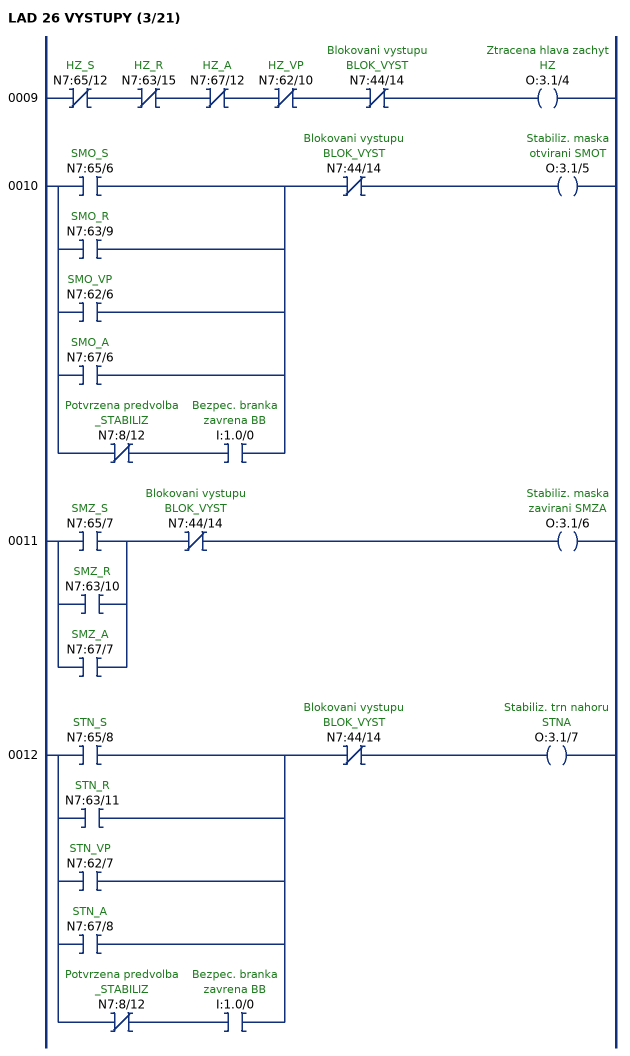
% Rung: 9 %
SOR XIO N7:65/12 XIO N7:63/15 XIO N7:67/12 XIO N7:62/10 XIO N7:44/14 OTE O:3.1/4 EOR
%   N7:65/12  HZ_S %
%   N7:63/15  HZ_R %
%   N7:67/12  HZ_A %
%   N7:62/10  HZ_VP %
%   N7:44/14  BLOK_VYST  "Blokovani vystupu" %
%   O:3.1/4  HZ  "Ztracena hlava zachyt" %
% Rung: 10 %
SOR BST XIC N7:65/6 NXB XIC N7:63/9 NXB XIC N7:62/6 NXB XIC N7:67/6 NXB XIO N7:8/12 XIC I:1.0/0 BND XIO N7:44/14 OTE O:3.1/5 EOR
%   N7:65/6  SMO_S %
%   N7:63/9  SMO_R %
%   N7:62/6  SMO_VP %
%   N7:67/6  SMO_A %
%   N7:8/12  _STABILIZ  "Potvrzena predvolba" %
%   I:1.0/0  BB  "Bezpec. branka zavrena" %
%   N7:44/14  BLOK_VYST  "Blokovani vystupu" %
%   O:3.1/5  SMOT  "Stabiliz. maska otvirani" %
% Rung: 11 %
SOR BST XIC N7:65/7 NXB XIC N7:63/10 NXB XIC N7:67/7 BND XIO N7:44/14 OTE O:3.1/6 EOR
%   N7:65/7  SMZ_S %
%   N7:63/10  SMZ_R %
%   N7:67/7  SMZ_A %
%   N7:44/14  BLOK_VYST  "Blokovani vystupu" %
%   O:3.1/6  SMZA  "Stabiliz. maska zavirani" %
% Rung: 12 %
SOR BST XIC N7:65/8 NXB XIC N7:63/11 NXB XIC N7:62/7 NXB XIC N7:67/8 NXB XIO N7:8/12 XIC I:1.0/0 BND XIO N7:44/14 OTE O:3.1/7 EOR
%   N7:65/8  STN_S %
%   N7:63/11  STN_R %
%   N7:62/7  STN_VP %
%   N7:67/8  STN_A %
%   N7:8/12  _STABILIZ  "Potvrzena predvolba" %
%   I:1.0/0  BB  "Bezpec. branka zavrena" %
%   N7:44/14  BLOK_VYST  "Blokovani vystupu" %
%   O:3.1/7  STNA  "Stabiliz. trn nahoru" %

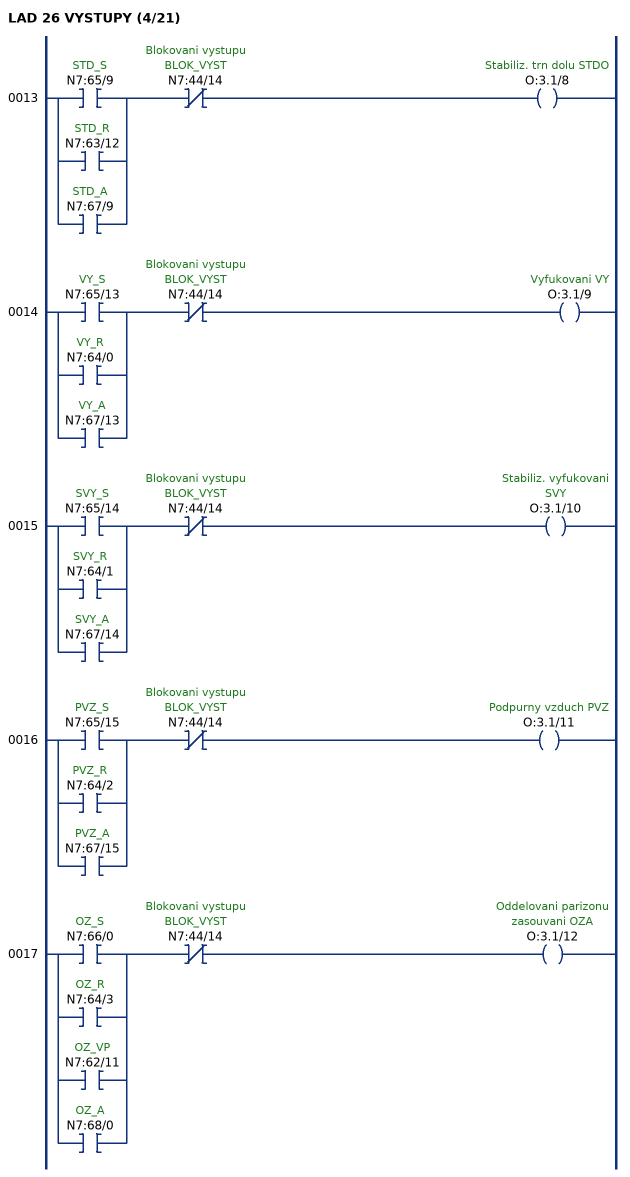
% Rung: 13 %
SOR BST XIC N7:65/9 NXB XIC N7:63/12 NXB XIC N7:67/9 BND XIO N7:44/14 OTE O:3.1/8 EOR
%   N7:65/9  STD_S %
%   N7:63/12  STD_R %
%   N7:67/9  STD_A %
%   N7:44/14  BLOK_VYST  "Blokovani vystupu" %
%   O:3.1/8  STDO  "Stabiliz. trn dolu" %
% Rung: 14 %
SOR BST XIC N7:65/13 NXB XIC N7:64/0 NXB XIC N7:67/13 BND XIO N7:44/14 OTE O:3.1/9 EOR
%   N7:65/13  VY_S %
%   N7:64/0  VY_R %
%   N7:67/13  VY_A %
%   N7:44/14  BLOK_VYST  "Blokovani vystupu" %
%   O:3.1/9  VY  "Vyfukovani" %
% Rung: 15 %
SOR BST XIC N7:65/14 NXB XIC N7:64/1 NXB XIC N7:67/14 BND XIO N7:44/14 OTE O:3.1/10 EOR
%   N7:65/14  SVY_S %
%   N7:64/1  SVY_R %
%   N7:67/14  SVY_A %
%   N7:44/14  BLOK_VYST  "Blokovani vystupu" %
%   O:3.1/10  SVY  "Stabiliz. vyfukovani" %
% Rung: 16 %
SOR BST XIC N7:65/15 NXB XIC N7:64/2 NXB XIC N7:67/15 BND XIO N7:44/14 OTE O:3.1/11 EOR
%   N7:65/15  PVZ_S %
%   N7:64/2  PVZ_R %
%   N7:67/15  PVZ_A %
%   N7:44/14  BLOK_VYST  "Blokovani vystupu" %
%   O:3.1/11  PVZ  "Podpurny vzduch" %
% Rung: 17 %
SOR BST XIC N7:66/0 NXB XIC N7:64/3 NXB XIC N7:62/11 NXB XIC N7:68/0 BND XIO N7:44/14 OTE O:3.1/12 EOR
%   N7:66/0  OZ_S %
%   N7:64/3  OZ_R %
%   N7:62/11  OZ_VP %
%   N7:68/0  OZ_A %
%   N7:44/14  BLOK_VYST  "Blokovani vystupu" %
%   O:3.1/12  OZA  "Oddelovani parizonu zasouvani" %

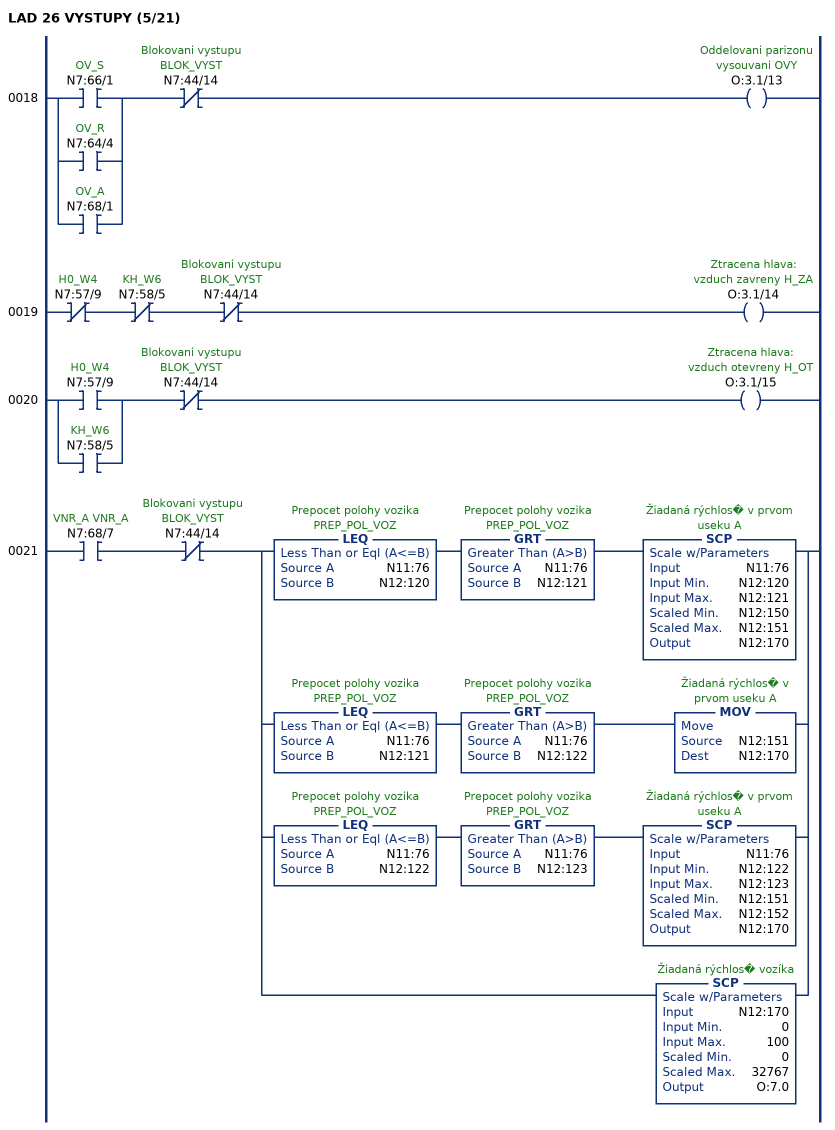
% Rung: 18 %
SOR BST XIC N7:66/1 NXB XIC N7:64/4 NXB XIC N7:68/1 BND XIO N7:44/14 OTE O:3.1/13 EOR
%   N7:66/1  OV_S %
%   N7:64/4  OV_R %
%   N7:68/1  OV_A %
%   N7:44/14  BLOK_VYST  "Blokovani vystupu" %
%   O:3.1/13  OVY  "Oddelovani parizonu vysouvani" %
% Rung: 19 %
SOR XIO N7:57/9 XIO N7:58/5 XIO N7:44/14 OTE O:3.1/14 EOR
%   N7:57/9  H0_W4 %
%   N7:58/5  KH_W6 %
%   N7:44/14  BLOK_VYST  "Blokovani vystupu" %
%   O:3.1/14  H_ZA  "Ztracena hlava: vzduch zavreny" %
% Rung: 20 %
SOR BST XIC N7:57/9 NXB XIC N7:58/5 BND XIO N7:44/14 OTE O:3.1/15 EOR
%   N7:57/9  H0_W4 %
%   N7:58/5  KH_W6 %
%   N7:44/14  BLOK_VYST  "Blokovani vystupu" %
%   O:3.1/15  H_OT  "Ztracena hlava: vzduch otevreny" %
% Rung: 21 %
SOR XIC N7:68/7 XIO N7:44/14 BST LEQ N11:76 N12:120 GRT N11:76 N12:121 SCP N11:76 N12:120 N12:121 N12:150 N12:151 N12:170 NXB LEQ N11:76 N12:121 GRT N11:76 N12:122 MOV N12:151 N12:170 NXB LEQ N11:76 N12:122 GRT N11:76 N12:123 SCP N11:76 N12:122 N12:123 N12:151 N12:152 N12:170 NXB SCP N12:170 0 100 0 32767 O:7.0 BND EOR
%   N7:68/7  VNR_A  "VNR_A" %
%   N7:44/14  BLOK_VYST  "Blokovani vystupu" %
%   N11:76  PREP_POL_VOZ  "Prepocet polohy vozika" %
%   N12:120  "Žiadana poloha vozika c.1 hore" %
%   N12:121  "Žiadana poloha vozika c.2 hore" %
%   N12:150  "Žiadaná rýchlost vozíka c.1 hore" %
%   N12:151  "Žiadaná rýchlost vozíka c.2 hore" %
%   N12:170  "Žiadaná rýchlos� v prvom useku A" %
%   N12:122  "Žiadana poloha vozika c.3 hore" %
%   N12:123  N123  "Žiadana poloha vozika c.4 hore" %
%   N12:152  "Žiadaná rýchlost vozíka c.3 hore" %
%   O:7.0  "Žiadaná rýchlos� vozíka" %

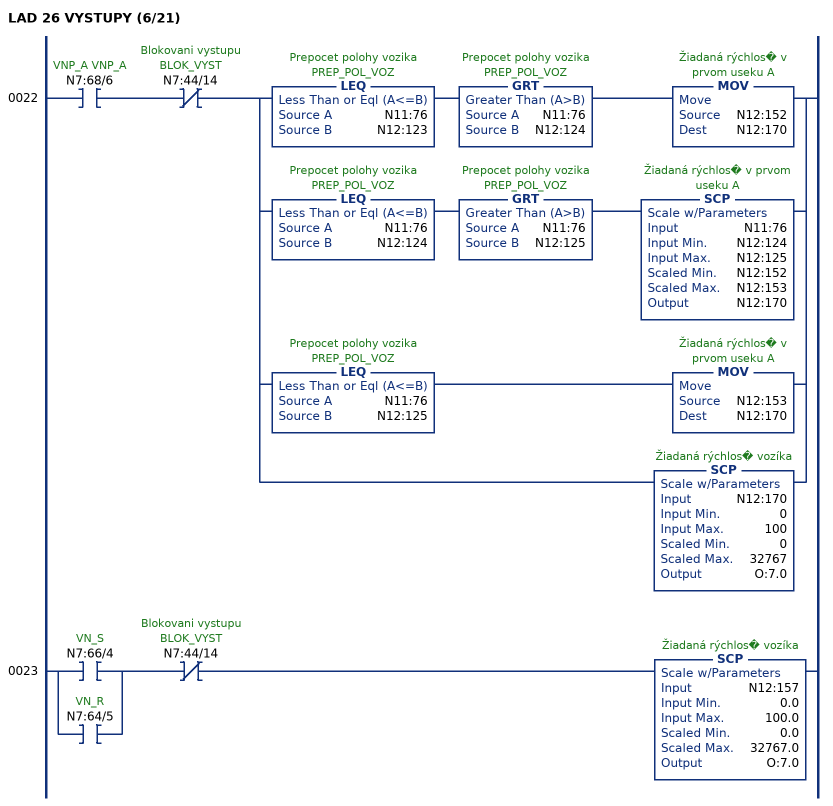
% Rung: 22 %
SOR XIC N7:68/6 XIO N7:44/14 BST LEQ N11:76 N12:123 GRT N11:76 N12:124 MOV N12:152 N12:170 NXB LEQ N11:76 N12:124 GRT N11:76 N12:125 SCP N11:76 N12:124 N12:125 N12:152 N12:153 N12:170 NXB LEQ N11:76 N12:125 MOV N12:153 N12:170 NXB SCP N12:170 0 100 0 32767 O:7.0 BND EOR
%   N7:68/6  VNP_A  "VNP_A" %
%   N7:44/14  BLOK_VYST  "Blokovani vystupu" %
%   N11:76  PREP_POL_VOZ  "Prepocet polohy vozika" %
%   N12:123  N123  "Žiadana poloha vozika c.4 hore" %
%   N12:124  "Žiadana poloha vozika c.5 hore" %
%   N12:152  "Žiadaná rýchlost vozíka c.3 hore" %
%   N12:170  "Žiadaná rýchlos� v prvom useku A" %
%   N12:125  "Žiadaná poloha c.3 vozík dole" %
%   N12:153  "Žiadaná rýchlost vozíka c.1 dolu" %
%   O:7.0  "Žiadaná rýchlos� vozíka" %
% Rung: 23 %
SOR BST XIC N7:66/4 NXB XIC N7:64/5 BND XIO N7:44/14 SCP N12:157 0.0 100.0 0.0 32767.0 O:7.0 EOR
%   N7:66/4  VN_S %
%   N7:64/5  VN_R %
%   N7:44/14  BLOK_VYST  "Blokovani vystupu" %
%   O:7.0  "Žiadaná rýchlos� vozíka" %

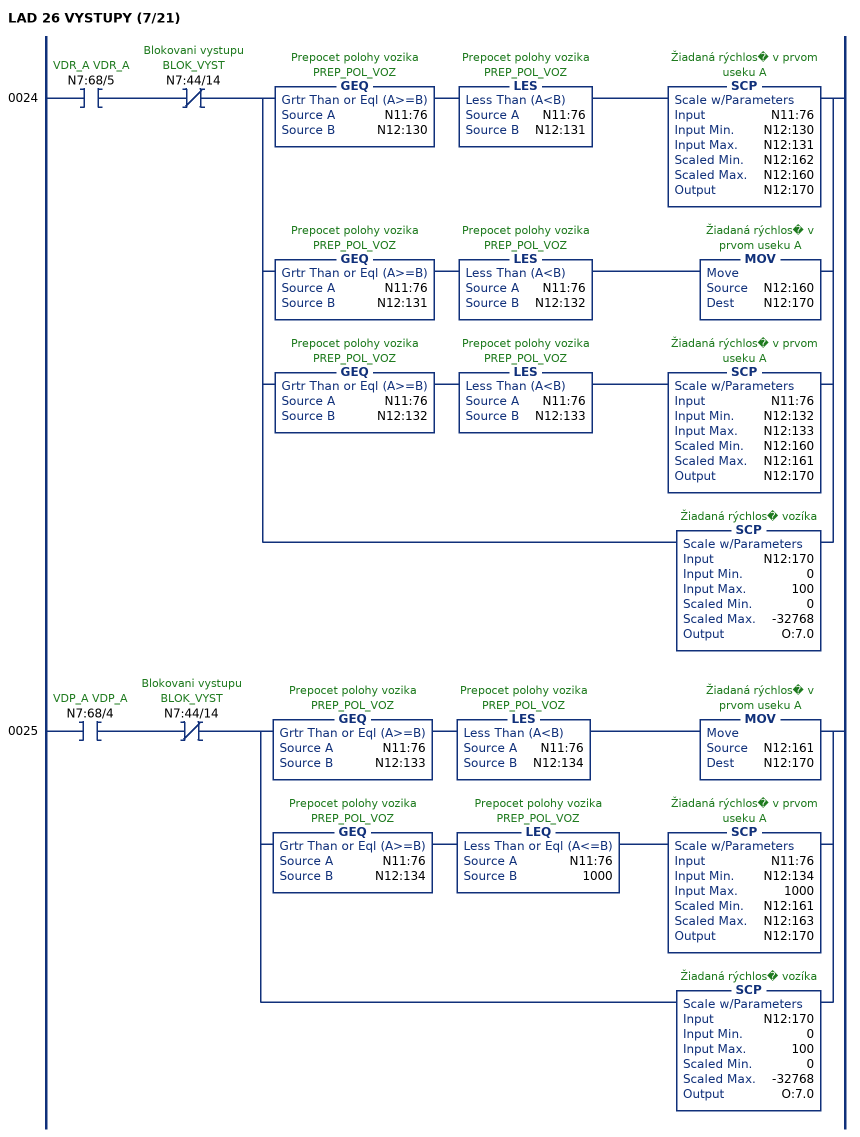
% Rung: 24 %
SOR XIC N7:68/5 XIO N7:44/14 BST GEQ N11:76 N12:130 LES N11:76 N12:131 SCP N11:76 N12:130 N12:131 N12:162 N12:160 N12:170 NXB GEQ N11:76 N12:131 LES N11:76 N12:132 MOV N12:160 N12:170 NXB GEQ N11:76 N12:132 LES N11:76 N12:133 SCP N11:76 N12:132 N12:133 N12:160 N12:161 N12:170 NXB SCP N12:170 0 100 0 -32768 O:7.0 BND EOR
%   N7:68/5  VDR_A  "VDR_A" %
%   N7:44/14  BLOK_VYST  "Blokovani vystupu" %
%   N11:76  PREP_POL_VOZ  "Prepocet polohy vozika" %
%   N12:170  "Žiadaná rýchlos� v prvom useku A" %
%   O:7.0  "Žiadaná rýchlos� vozíka" %
% Rung: 25 %
SOR XIC N7:68/4 XIO N7:44/14 BST GEQ N11:76 N12:133 LES N11:76 N12:134 MOV N12:161 N12:170 NXB GEQ N11:76 N12:134 LEQ N11:76 1000 SCP N11:76 N12:134 1000 N12:161 N12:163 N12:170 NXB SCP N12:170 0 100 0 -32768 O:7.0 BND EOR
%   N7:68/4  VDP_A  "VDP_A" %
%   N7:44/14  BLOK_VYST  "Blokovani vystupu" %
%   N11:76  PREP_POL_VOZ  "Prepocet polohy vozika" %
%   N12:170  "Žiadaná rýchlos� v prvom useku A" %
%   O:7.0  "Žiadaná rýchlos� vozíka" %

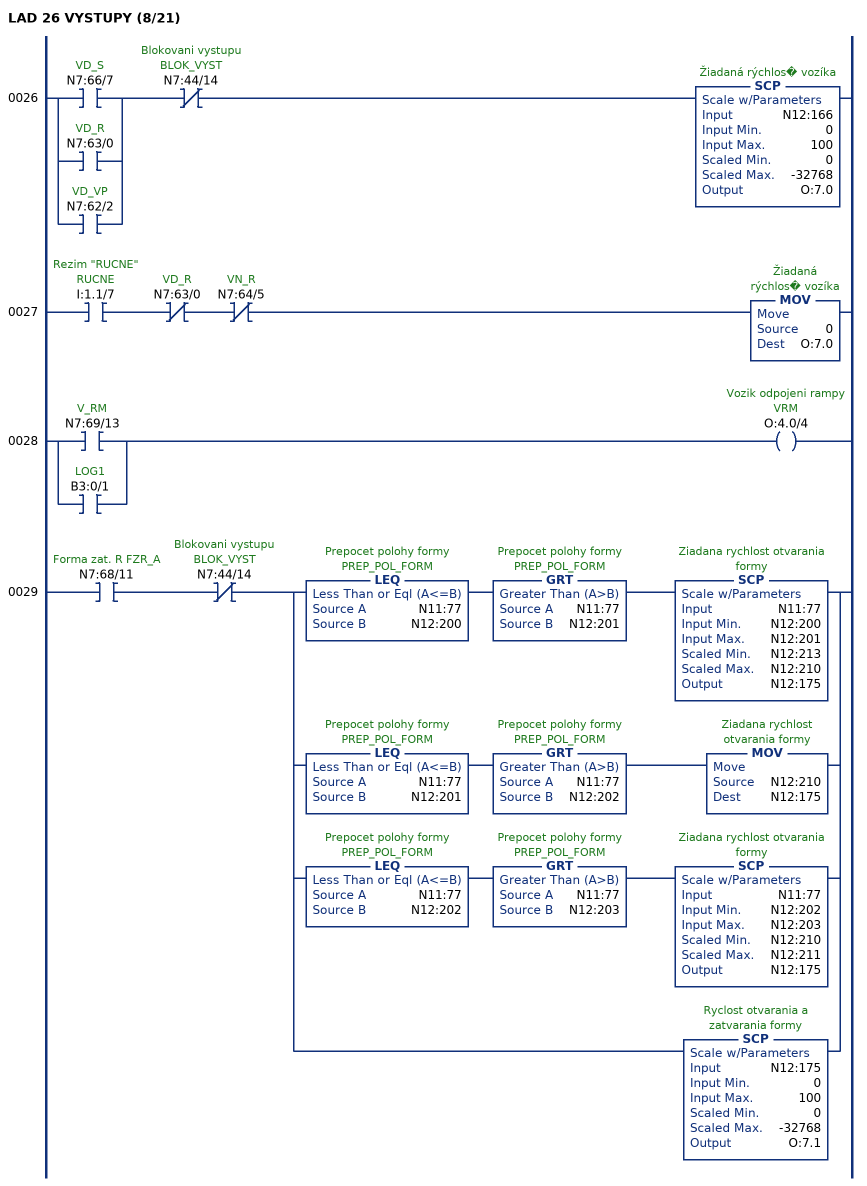
% Rung: 26 %
SOR BST XIC N7:66/7 NXB XIC N7:63/0 NXB XIC N7:62/2 BND XIO N7:44/14 SCP N12:166 0 100 0 -32768 O:7.0 EOR
%   N7:66/7  VD_S %
%   N7:63/0  VD_R %
%   N7:62/2  VD_VP %
%   N7:44/14  BLOK_VYST  "Blokovani vystupu" %
%   O:7.0  "Žiadaná rýchlos� vozíka" %
% Rung: 27 %
SOR XIC I:1.1/7 XIO N7:63/0 XIO N7:64/5 MOV 0 O:7.0 EOR
%   I:1.1/7  RUCNE  "Rezim "RUCNE"" %
%   N7:63/0  VD_R %
%   N7:64/5  VN_R %
%   O:7.0  "Žiadaná rýchlos� vozíka" %
% Rung: 28 %
SOR BST XIC N7:69/13 NXB XIC B3:0/1 BND OTE O:4.0/4 EOR
%   N7:69/13  V_RM %
%   B3:0/1  LOG1 %
%   O:4.0/4  VRM  "Vozik odpojeni rampy" %
% Rung: 29 %
SOR XIC N7:68/11 XIO N7:44/14 BST LEQ N11:77 N12:200 GRT N11:77 N12:201 SCP N11:77 N12:200 N12:201 N12:213 N12:210 N12:175 NXB LEQ N11:77 N12:201 GRT N11:77 N12:202 MOV N12:210 N12:175 NXB LEQ N11:77 N12:202 GRT N11:77 N12:203 SCP N11:77 N12:202 N12:203 N12:210 N12:211 N12:175 NXB SCP N12:175 0 100 0 -32768 O:7.1 BND EOR
%   N7:68/11  FZR_A  "Forma zat. R" %
%   N7:44/14  BLOK_VYST  "Blokovani vystupu" %
%   N11:77  PREP_POL_FORM  "Prepocet polohy formy" %
%   N12:175  "Ziadana rychlost otvarania formy" %
%   O:7.1  "Ryclost otvarania a zatvarania formy" %

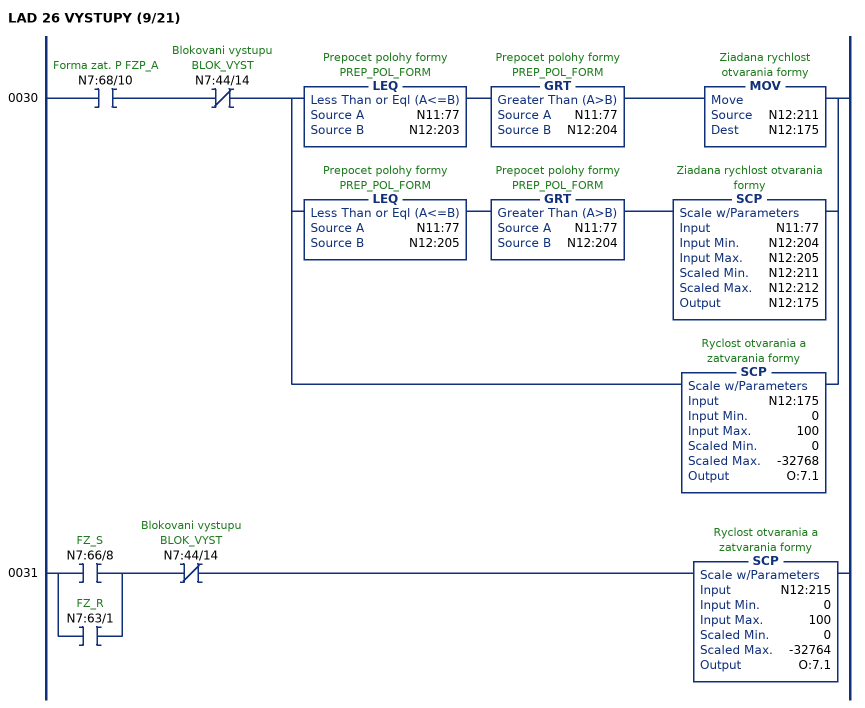
% Rung: 30 %
SOR XIC N7:68/10 XIO N7:44/14 BST LEQ N11:77 N12:203 GRT N11:77 N12:204 MOV N12:211 N12:175 NXB LEQ N11:77 N12:205 GRT N11:77 N12:204 SCP N11:77 N12:204 N12:205 N12:211 N12:212 N12:175 NXB SCP N12:175 0 100 0 -32768 O:7.1 BND EOR
%   N7:68/10  FZP_A  "Forma zat. P" %
%   N7:44/14  BLOK_VYST  "Blokovani vystupu" %
%   N11:77  PREP_POL_FORM  "Prepocet polohy formy" %
%   N12:175  "Ziadana rychlost otvarania formy" %
%   O:7.1  "Ryclost otvarania a zatvarania formy" %
% Rung: 31 %
SOR BST XIC N7:66/8 NXB XIC N7:63/1 BND XIO N7:44/14 SCP N12:215 0 100 0 -32764 O:7.1 EOR
%   N7:66/8  FZ_S %
%   N7:63/1  FZ_R %
%   N7:44/14  BLOK_VYST  "Blokovani vystupu" %
%   O:7.1  "Ryclost otvarania a zatvarania formy" %

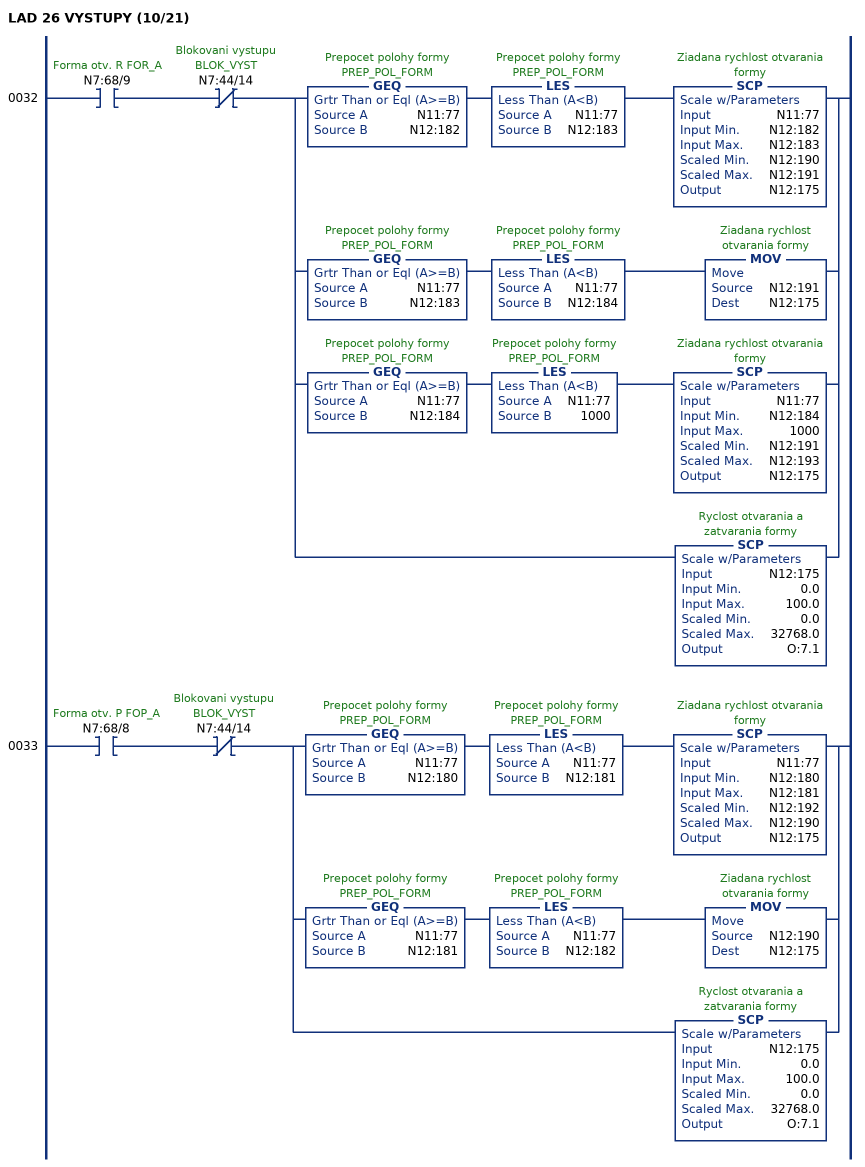
% Rung: 32 %
SOR XIC N7:68/9 XIO N7:44/14 BST GEQ N11:77 N12:182 LES N11:77 N12:183 SCP N11:77 N12:182 N12:183 N12:190 N12:191 N12:175 NXB GEQ N11:77 N12:183 LES N11:77 N12:184 MOV N12:191 N12:175 NXB GEQ N11:77 N12:184 LES N11:77 1000 SCP N11:77 N12:184 1000 N12:191 N12:193 N12:175 NXB SCP N12:175 0.0 100.0 0.0 32768.0 O:7.1 BND EOR
%   N7:68/9  FOR_A  "Forma otv. R" %
%   N7:44/14  BLOK_VYST  "Blokovani vystupu" %
%   N11:77  PREP_POL_FORM  "Prepocet polohy formy" %
%   N12:190  "Ziadana ryhlost otvarania formy v prvom useku" %
%   N12:191  "Ziadana ryhlost otvarania formy v druhom useku" %
%   N12:175  "Ziadana rychlost otvarania formy" %
%   O:7.1  "Ryclost otvarania a zatvarania formy" %
% Rung: 33 %
SOR XIC N7:68/8 XIO N7:44/14 BST GEQ N11:77 N12:180 LES N11:77 N12:181 SCP N11:77 N12:180 N12:181 N12:192 N12:190 N12:175 NXB GEQ N11:77 N12:181 LES N11:77 N12:182 MOV N12:190 N12:175 NXB SCP N12:175 0.0 100.0 0.0 32768.0 O:7.1 BND EOR
%   N7:68/8  FOP_A  "Forma otv. P" %
%   N7:44/14  BLOK_VYST  "Blokovani vystupu" %
%   N11:77  PREP_POL_FORM  "Prepocet polohy formy" %
%   N12:190  "Ziadana ryhlost otvarania formy v prvom useku" %
%   N12:175  "Ziadana rychlost otvarania formy" %
%   O:7.1  "Ryclost otvarania a zatvarania formy" %

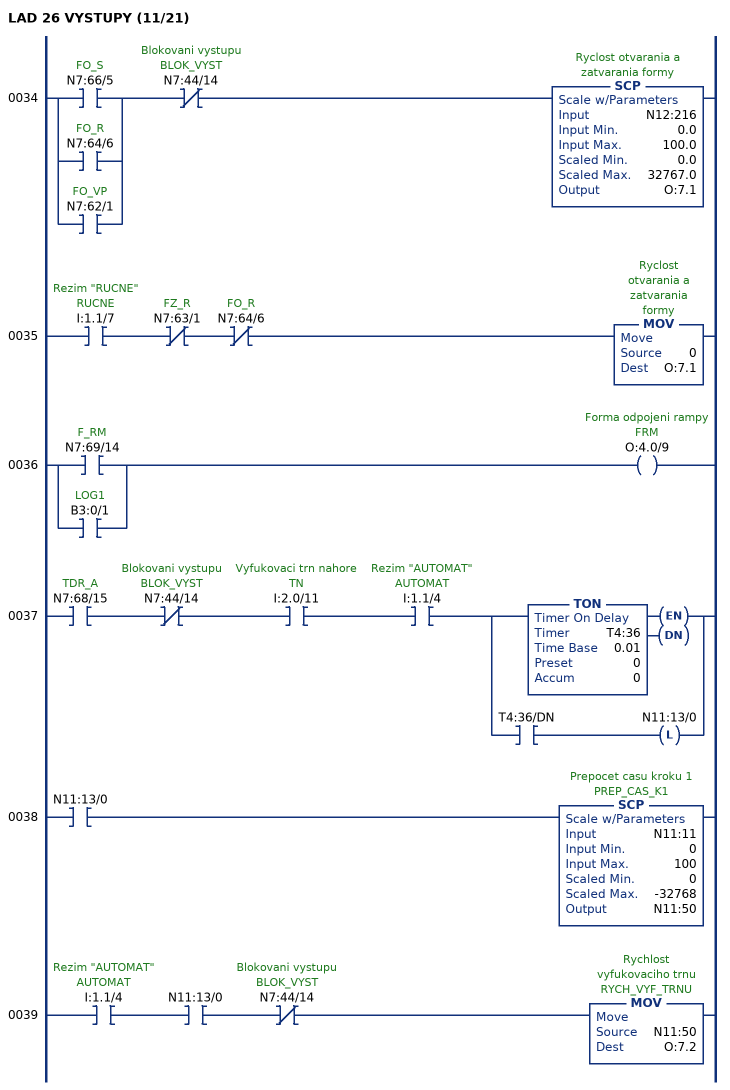
% Rung: 34 %
SOR BST XIC N7:66/5 NXB XIC N7:64/6 NXB XIC N7:62/1 BND XIO N7:44/14 SCP N12:216 0.0 100.0 0.0 32767.0 O:7.1 EOR
%   N7:66/5  FO_S %
%   N7:64/6  FO_R %
%   N7:62/1  FO_VP %
%   N7:44/14  BLOK_VYST  "Blokovani vystupu" %
%   O:7.1  "Ryclost otvarania a zatvarania formy" %
% Rung: 35 %
SOR XIC I:1.1/7 XIO N7:63/1 XIO N7:64/6 MOV 0 O:7.1 EOR
%   I:1.1/7  RUCNE  "Rezim "RUCNE"" %
%   N7:63/1  FZ_R %
%   N7:64/6  FO_R %
%   O:7.1  "Ryclost otvarania a zatvarania formy" %
% Rung: 36 %
SOR BST XIC N7:69/14 NXB XIC B3:0/1 BND OTE O:4.0/9 EOR
%   N7:69/14  F_RM %
%   B3:0/1  LOG1 %
%   O:4.0/9  FRM  "Forma odpojeni rampy" %
% Rung: 37 %
SOR XIC N7:68/15 XIO N7:44/14 XIC I:2.0/11 XIC I:1.1/4 BST TON T4:36 0.01 0 0 NXB XIC T4:36/DN OTL N11:13/0 BND EOR
%   N7:68/15  TDR_A %
%   N7:44/14  BLOK_VYST  "Blokovani vystupu" %
%   I:2.0/11  TN  "Vyfukovaci trn nahore" %
%   I:1.1/4  AUTOMAT  "Rezim "AUTOMAT"" %
% Rung: 38 %
SOR XIC N11:13/0 SCP N11:11 0 100 0 -32768 N11:50 EOR
%   N11:11  CAS_K1  "Cas kroku 1" %
%   N11:50  PREP_CAS_K1  "Prepocet casu kroku 1" %
% Rung: 39 %
SOR XIC I:1.1/4 XIC N11:13/0 XIO N7:44/14 MOV N11:50 O:7.2 EOR
%   I:1.1/4  AUTOMAT  "Rezim "AUTOMAT"" %
%   N7:44/14  BLOK_VYST  "Blokovani vystupu" %
%   N11:50  PREP_CAS_K1  "Prepocet casu kroku 1" %
%   O:7.2  RYCH_VYF_TRNU  "Rychlost vyfukovaciho trnu" %

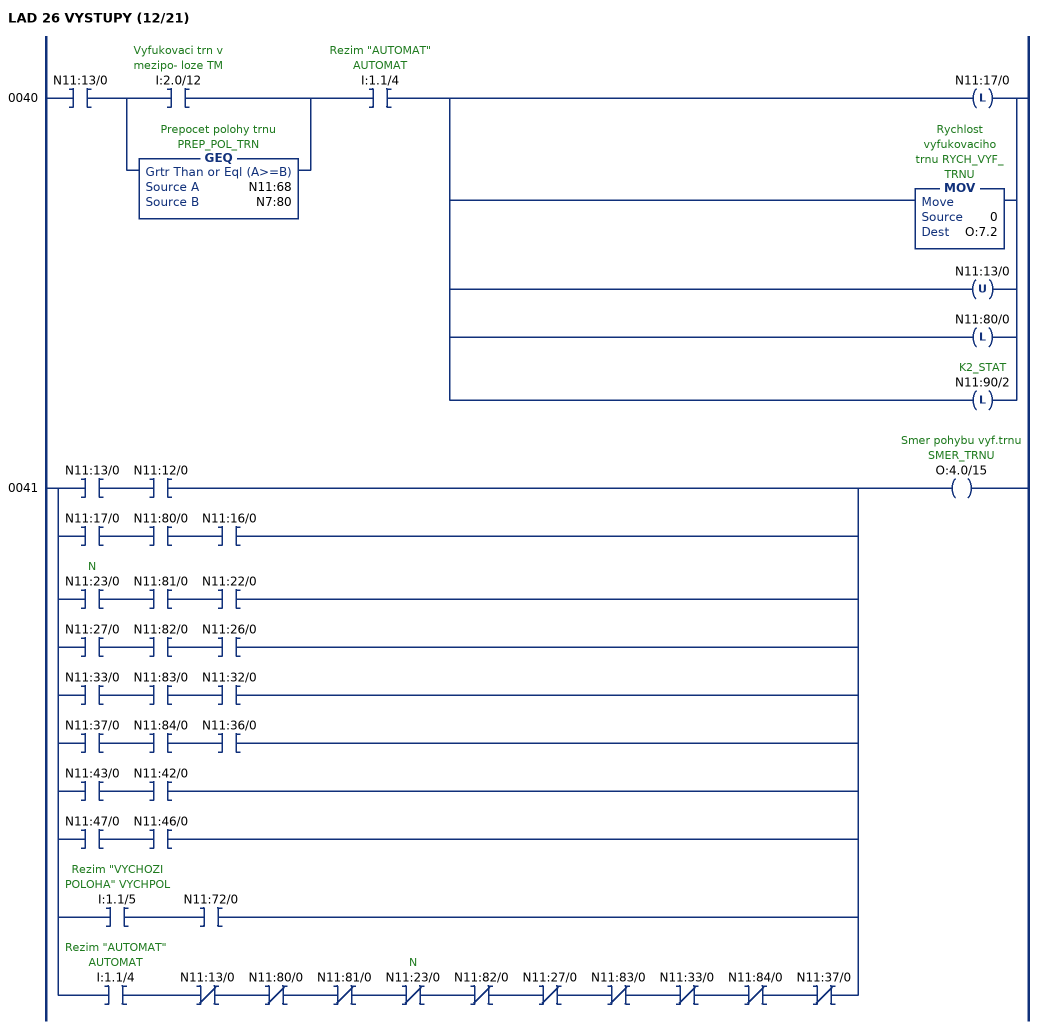
% Rung: 40 %
SOR XIC N11:13/0 BST XIC I:2.0/12 NXB GEQ N11:68 N7:80 BND XIC I:1.1/4 BST OTL N11:17/0 NXB MOV 0 O:7.2 NXB OTU N11:13/0 NXB OTL N11:80/0 NXB OTL N11:90/2 BND EOR
%   I:2.0/12  TM  "Vyfukovaci trn v mezipo- loze" %
%   N11:68  PREP_POL_TRN  "Prepocet polohy trnu" %
%   I:1.1/4  AUTOMAT  "Rezim "AUTOMAT"" %
%   O:7.2  RYCH_VYF_TRNU  "Rychlost vyfukovaciho trnu" %
%   N11:90/2  K2_STAT %
% Rung: 41 %
SOR BST XIC N11:13/0 XIC N11:12/0 NXB XIC N11:17/0 XIC N11:80/0 XIC N11:16/0 NXB XIC N11:23/0 XIC N11:81/0 XIC N11:22/0 NXB XIC N11:27/0 XIC N11:82/0 XIC N11:26/0 NXB XIC N11:33/0 XIC N11:83/0 XIC N11:32/0 NXB XIC N11:37/0 XIC N11:84/0 XIC N11:36/0 NXB XIC N11:43/0 XIC N11:42/0 NXB XIC N11:47/0 XIC N11:46/0 NXB XIC I:1.1/5 XIC N11:72/0 NXB XIC I:1.1/4 XIO N11:13/0 XIO N11:80/0 XIO N11:81/0 XIO N11:23/0 XIO N11:82/0 XIO N11:27/0 XIO N11:83/0 XIO N11:33/0 XIO N11:84/0 XIO N11:37/0 BND OTE O:4.0/15 EOR
%   N11:23/0  N %
%   I:1.1/5  VYCHPOL  "Rezim "VYCHOZI POLOHA"" %
%   I:1.1/4  AUTOMAT  "Rezim "AUTOMAT"" %
%   O:4.0/15  SMER_TRNU  "Smer pohybu vyf.trnu" %

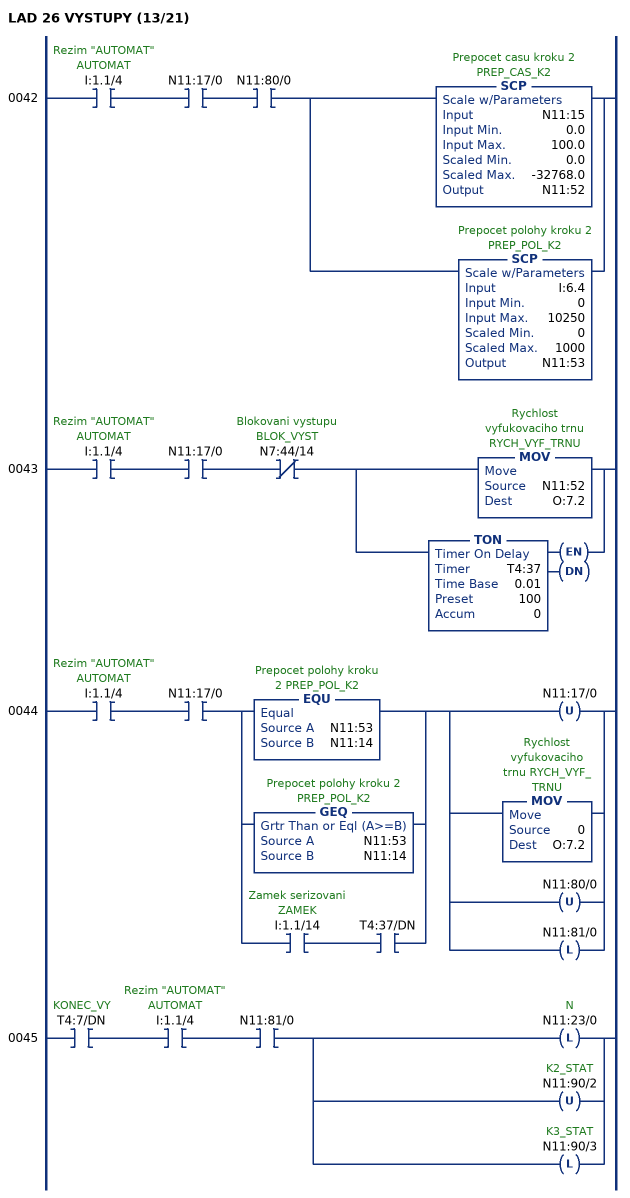
% Rung: 42 %
SOR XIC I:1.1/4 XIC N11:17/0 XIC N11:80/0 BST SCP N11:15 0.0 100.0 0.0 -32768.0 N11:52 NXB SCP I:6.4 0 10250 0 1000 N11:53 BND EOR
%   I:1.1/4  AUTOMAT  "Rezim "AUTOMAT"" %
%   N11:15  CAS_K2  "Cas kroku 2" %
%   N11:52  PREP_CAS_K2  "Prepocet casu kroku 2" %
%   I:6.4  POL_VYF_TRNU  "Poloha vyfukovaciho trnu" %
%   N11:53  PREP_POL_K2  "Prepocet polohy kroku 2" %
% Rung: 43 %
SOR XIC I:1.1/4 XIC N11:17/0 XIO N7:44/14 BST MOV N11:52 O:7.2 NXB TON T4:37 0.01 100 0 BND EOR
%   I:1.1/4  AUTOMAT  "Rezim "AUTOMAT"" %
%   N7:44/14  BLOK_VYST  "Blokovani vystupu" %
%   N11:52  PREP_CAS_K2  "Prepocet casu kroku 2" %
%   O:7.2  RYCH_VYF_TRNU  "Rychlost vyfukovaciho trnu" %
% Rung: 44 %
SOR XIC I:1.1/4 XIC N11:17/0 BST EQU N11:53 N11:14 NXB GEQ N11:53 N11:14 NXB XIC I:1.1/14 XIC T4:37/DN BND BST OTU N11:17/0 NXB MOV 0 O:7.2 NXB OTU N11:80/0 NXB OTL N11:81/0 BND EOR
%   I:1.1/4  AUTOMAT  "Rezim "AUTOMAT"" %
%   N11:53  PREP_POL_K2  "Prepocet polohy kroku 2" %
%   N11:14  DR_K2  "Draha kroku 2" %
%   I:1.1/14  ZAMEK  "Zamek serizovani" %
%   O:7.2  RYCH_VYF_TRNU  "Rychlost vyfukovaciho trnu" %
% Rung: 45 %
SOR XIC T4:7/DN XIC I:1.1/4 XIC N11:81/0 BST OTL N11:23/0 NXB OTU N11:90/2 NXB OTL N11:90/3 BND EOR
%   T4:7/DN  KONEC_VY %
%   I:1.1/4  AUTOMAT  "Rezim "AUTOMAT"" %
%   N11:23/0  N %
%   N11:90/2  K2_STAT %
%   N11:90/3  K3_STAT %

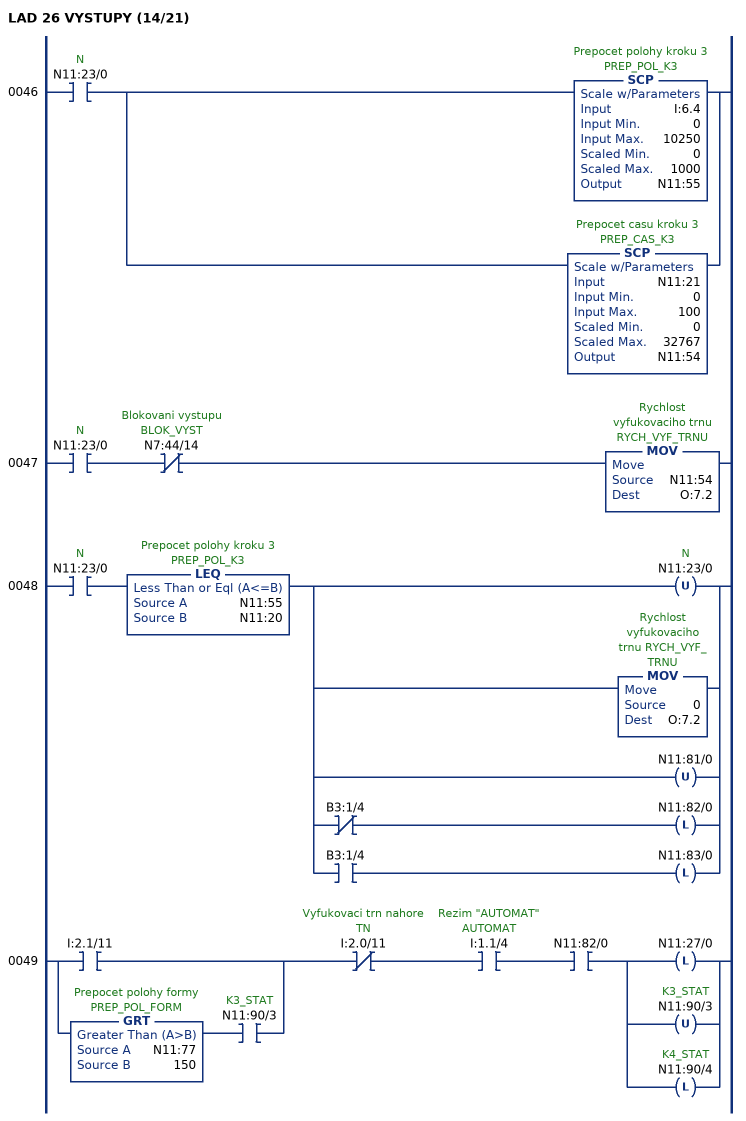
% Rung: 46 %
SOR XIC N11:23/0 BST SCP I:6.4 0 10250 0 1000 N11:55 NXB SCP N11:21 0 100 0 32767 N11:54 BND EOR
%   N11:23/0  N %
%   I:6.4  POL_VYF_TRNU  "Poloha vyfukovaciho trnu" %
%   N11:55  PREP_POL_K3  "Prepocet polohy kroku 3" %
%   N11:21  CAS_K3  "Cas kroku 3" %
%   N11:54  PREP_CAS_K3  "Prepocet casu kroku 3" %
% Rung: 47 %
SOR XIC N11:23/0 XIO N7:44/14 MOV N11:54 O:7.2 EOR
%   N11:23/0  N %
%   N7:44/14  BLOK_VYST  "Blokovani vystupu" %
%   N11:54  PREP_CAS_K3  "Prepocet casu kroku 3" %
%   O:7.2  RYCH_VYF_TRNU  "Rychlost vyfukovaciho trnu" %
% Rung: 48 %
SOR XIC N11:23/0 LEQ N11:55 N11:20 BST OTU N11:23/0 NXB MOV 0 O:7.2 NXB OTU N11:81/0 NXB XIO B3:1/4 OTL N11:82/0 NXB XIC B3:1/4 OTL N11:83/0 BND EOR
%   N11:23/0  N %
%   N11:55  PREP_POL_K3  "Prepocet polohy kroku 3" %
%   N11:20  DR_K3  "Draha kroku 3" %
%   O:7.2  RYCH_VYF_TRNU  "Rychlost vyfukovaciho trnu" %
% Rung: 49 %
SOR BST XIC I:2.1/11 NXB GRT N11:77 150 XIC N11:90/3 BND XIO I:2.0/11 XIC I:1.1/4 XIC N11:82/0 BST OTL N11:27/0 NXB OTU N11:90/3 NXB OTL N11:90/4 BND EOR
%   N11:77  PREP_POL_FORM  "Prepocet polohy formy" %
%   N11:90/3  K3_STAT %
%   I:2.0/11  TN  "Vyfukovaci trn nahore" %
%   I:1.1/4  AUTOMAT  "Rezim "AUTOMAT"" %
%   N11:90/4  K4_STAT %

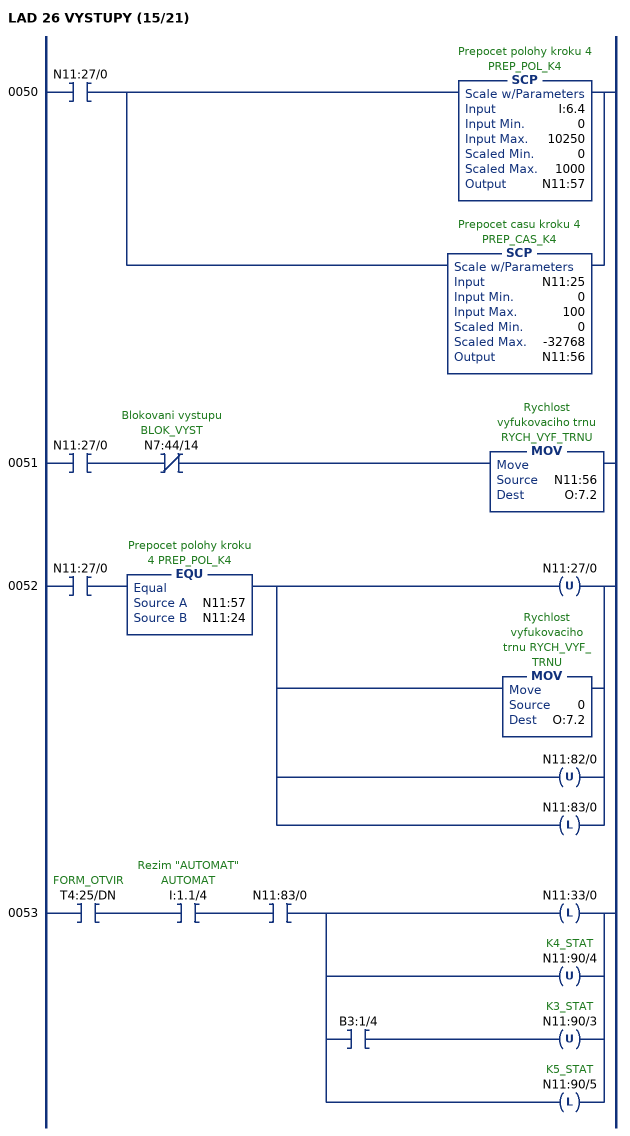
% Rung: 50 %
SOR XIC N11:27/0 BST SCP I:6.4 0 10250 0 1000 N11:57 NXB SCP N11:25 0 100 0 -32768 N11:56 BND EOR
%   I:6.4  POL_VYF_TRNU  "Poloha vyfukovaciho trnu" %
%   N11:57  PREP_POL_K4  "Prepocet polohy kroku 4" %
%   N11:25  CAS_K4  "Cas kroku 4" %
%   N11:56  PREP_CAS_K4  "Prepocet casu kroku 4" %
% Rung: 51 %
SOR XIC N11:27/0 XIO N7:44/14 MOV N11:56 O:7.2 EOR
%   N7:44/14  BLOK_VYST  "Blokovani vystupu" %
%   N11:56  PREP_CAS_K4  "Prepocet casu kroku 4" %
%   O:7.2  RYCH_VYF_TRNU  "Rychlost vyfukovaciho trnu" %
% Rung: 52 %
SOR XIC N11:27/0 EQU N11:57 N11:24 BST OTU N11:27/0 NXB MOV 0 O:7.2 NXB OTU N11:82/0 NXB OTL N11:83/0 BND EOR
%   N11:57  PREP_POL_K4  "Prepocet polohy kroku 4" %
%   N11:24  DR_K4  "Draha kroku 4" %
%   O:7.2  RYCH_VYF_TRNU  "Rychlost vyfukovaciho trnu" %
% Rung: 53 %
SOR XIC T4:25/DN XIC I:1.1/4 XIC N11:83/0 BST OTL N11:33/0 NXB OTU N11:90/4 NXB XIC B3:1/4 OTU N11:90/3 NXB OTL N11:90/5 BND EOR
%   T4:25/DN  FORM_OTVIR %
%   I:1.1/4  AUTOMAT  "Rezim "AUTOMAT"" %
%   N11:90/4  K4_STAT %
%   N11:90/3  K3_STAT %
%   N11:90/5  K5_STAT %

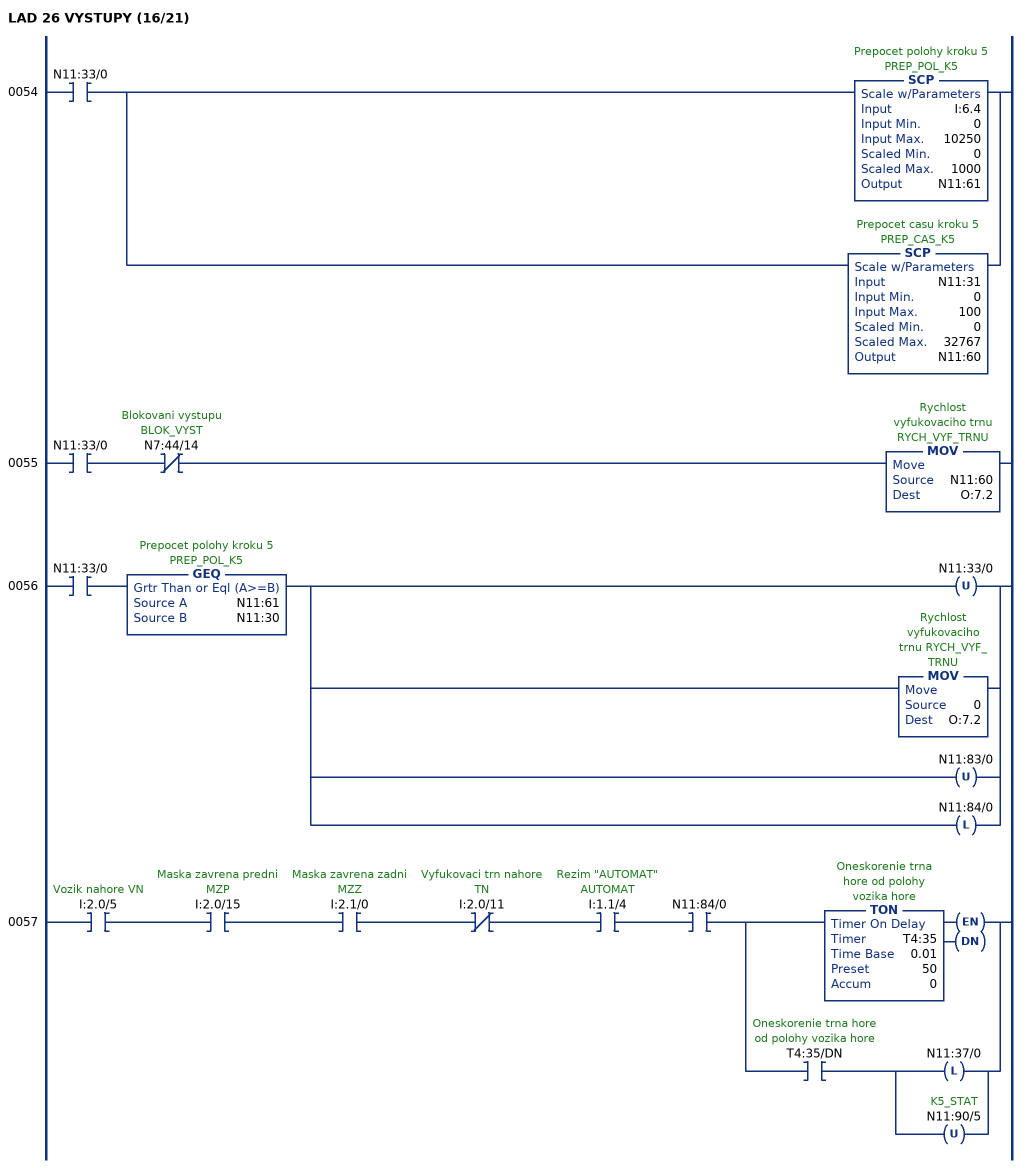
% Rung: 54 %
SOR XIC N11:33/0 BST SCP I:6.4 0 10250 0 1000 N11:61 NXB SCP N11:31 0 100 0 32767 N11:60 BND EOR
%   I:6.4  POL_VYF_TRNU  "Poloha vyfukovaciho trnu" %
%   N11:61  PREP_POL_K5  "Prepocet polohy kroku 5" %
%   N11:31  CAS_K5  "Cas kroku 5" %
%   N11:60  PREP_CAS_K5  "Prepocet casu kroku 5" %
% Rung: 55 %
SOR XIC N11:33/0 XIO N7:44/14 MOV N11:60 O:7.2 EOR
%   N7:44/14  BLOK_VYST  "Blokovani vystupu" %
%   N11:60  PREP_CAS_K5  "Prepocet casu kroku 5" %
%   O:7.2  RYCH_VYF_TRNU  "Rychlost vyfukovaciho trnu" %
% Rung: 56 %
SOR XIC N11:33/0 GEQ N11:61 N11:30 BST OTU N11:33/0 NXB MOV 0 O:7.2 NXB OTU N11:83/0 NXB OTL N11:84/0 BND EOR
%   N11:61  PREP_POL_K5  "Prepocet polohy kroku 5" %
%   N11:30  DR_K5  "Draha kroku 5" %
%   O:7.2  RYCH_VYF_TRNU  "Rychlost vyfukovaciho trnu" %
% Rung: 57 %
SOR XIC I:2.0/5 XIC I:2.0/15 XIC I:2.1/0 XIO I:2.0/11 XIC I:1.1/4 XIC N11:84/0 BST TON T4:35 0.01 50 0 NXB XIC T4:35/DN BST OTL N11:37/0 NXB OTU N11:90/5 BND BND EOR
%   I:2.0/5  VN  "Vozik nahore" %
%   I:2.0/15  MZP  "Maska zavrena predni" %
%   I:2.1/0  MZZ  "Maska zavrena zadni" %
%   I:2.0/11  TN  "Vyfukovaci trn nahore" %
%   I:1.1/4  AUTOMAT  "Rezim "AUTOMAT"" %
%   T4:35  "Oneskorenie trna hore od polohy vozika hore" %
%   N11:90/5  K5_STAT %

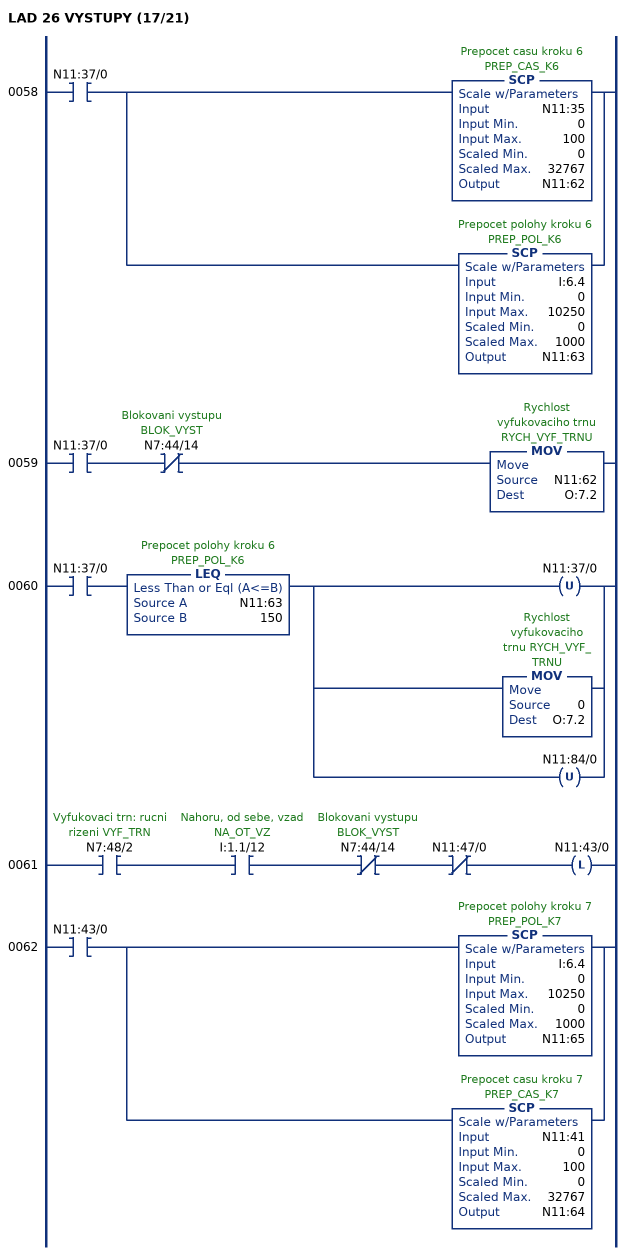
% Rung: 58 %
SOR XIC N11:37/0 BST SCP N11:35 0 100 0 32767 N11:62 NXB SCP I:6.4 0 10250 0 1000 N11:63 BND EOR
%   N11:35  CAS_K6  "Cas kroku 6" %
%   N11:62  PREP_CAS_K6  "Prepocet casu kroku 6" %
%   I:6.4  POL_VYF_TRNU  "Poloha vyfukovaciho trnu" %
%   N11:63  PREP_POL_K6  "Prepocet polohy kroku 6" %
% Rung: 59 %
SOR XIC N11:37/0 XIO N7:44/14 MOV N11:62 O:7.2 EOR
%   N7:44/14  BLOK_VYST  "Blokovani vystupu" %
%   N11:62  PREP_CAS_K6  "Prepocet casu kroku 6" %
%   O:7.2  RYCH_VYF_TRNU  "Rychlost vyfukovaciho trnu" %
% Rung: 60 %
SOR XIC N11:37/0 LEQ N11:63 150 BST OTU N11:37/0 NXB MOV 0 O:7.2 NXB OTU N11:84/0 BND EOR
%   N11:63  PREP_POL_K6  "Prepocet polohy kroku 6" %
%   O:7.2  RYCH_VYF_TRNU  "Rychlost vyfukovaciho trnu" %
% Rung: 61 %
SOR XIC N7:48/2 XIC I:1.1/12 XIO N7:44/14 XIO N11:47/0 OTL N11:43/0 EOR
%   N7:48/2  VYF_TRN  "Vyfukovaci trn: rucni rizeni" %
%   I:1.1/12  NA_OT_VZ  "Nahoru, od sebe, vzad" %
%   N7:44/14  BLOK_VYST  "Blokovani vystupu" %
% Rung: 62 %
SOR XIC N11:43/0 BST SCP I:6.4 0 10250 0 1000 N11:65 NXB SCP N11:41 0 100 0 32767 N11:64 BND EOR
%   I:6.4  POL_VYF_TRNU  "Poloha vyfukovaciho trnu" %
%   N11:65  PREP_POL_K7  "Prepocet polohy kroku 7" %
%   N11:41  CAS_K7  "Cas kroku 7" %
%   N11:64  PREP_CAS_K7  "Prepocet casu kroku 7" %

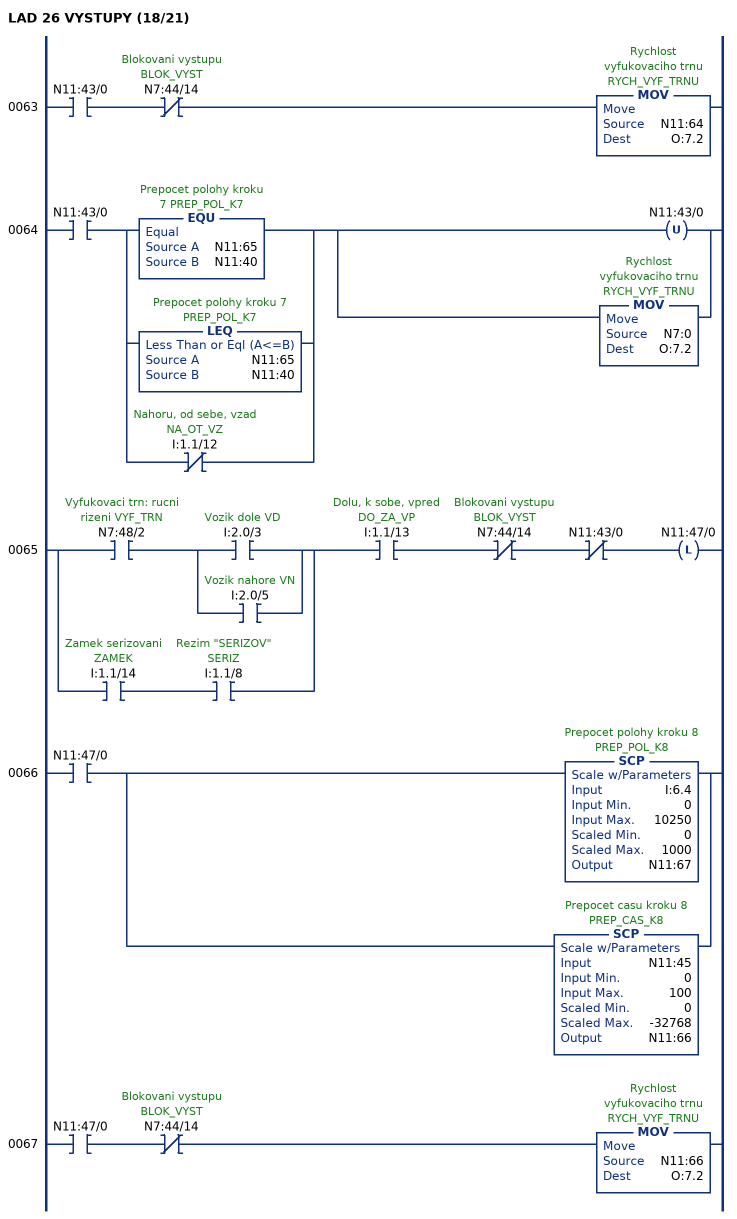
% Rung: 63 %
SOR XIC N11:43/0 XIO N7:44/14 MOV N11:64 O:7.2 EOR
%   N7:44/14  BLOK_VYST  "Blokovani vystupu" %
%   N11:64  PREP_CAS_K7  "Prepocet casu kroku 7" %
%   O:7.2  RYCH_VYF_TRNU  "Rychlost vyfukovaciho trnu" %
% Rung: 64 %
SOR XIC N11:43/0 BST EQU N11:65 N11:40 NXB LEQ N11:65 N11:40 NXB XIO I:1.1/12 BND BST OTU N11:43/0 NXB MOV N7:0 O:7.2 BND EOR
%   N11:65  PREP_POL_K7  "Prepocet polohy kroku 7" %
%   N11:40  DR_K7  "Draha kroku 7" %
%   I:1.1/12  NA_OT_VZ  "Nahoru, od sebe, vzad" %
%   O:7.2  RYCH_VYF_TRNU  "Rychlost vyfukovaciho trnu" %
% Rung: 65 %
SOR BST XIC N7:48/2 BST XIC I:2.0/3 NXB XIC I:2.0/5 BND NXB XIC I:1.1/14 XIC I:1.1/8 BND XIC I:1.1/13 XIO N7:44/14 XIO N11:43/0 OTL N11:47/0 EOR
%   N7:48/2  VYF_TRN  "Vyfukovaci trn: rucni rizeni" %
%   I:2.0/3  VD  "Vozik dole" %
%   I:2.0/5  VN  "Vozik nahore" %
%   I:1.1/14  ZAMEK  "Zamek serizovani" %
%   I:1.1/8  SERIZ  "Rezim "SERIZOV"" %
%   I:1.1/13  DO_ZA_VP  "Dolu, k sobe, vpred" %
%   N7:44/14  BLOK_VYST  "Blokovani vystupu" %
% Rung: 66 %
SOR XIC N11:47/0 BST SCP I:6.4 0 10250 0 1000 N11:67 NXB SCP N11:45 0 100 0 -32768 N11:66 BND EOR
%   I:6.4  POL_VYF_TRNU  "Poloha vyfukovaciho trnu" %
%   N11:67  PREP_POL_K8  "Prepocet polohy kroku 8" %
%   N11:45  CAS_K8  "Cas kroku 8" %
%   N11:66  PREP_CAS_K8  "Prepocet casu kroku 8" %
% Rung: 67 %
SOR XIC N11:47/0 XIO N7:44/14 MOV N11:66 O:7.2 EOR
%   N7:44/14  BLOK_VYST  "Blokovani vystupu" %
%   N11:66  PREP_CAS_K8  "Prepocet casu kroku 8" %
%   O:7.2  RYCH_VYF_TRNU  "Rychlost vyfukovaciho trnu" %

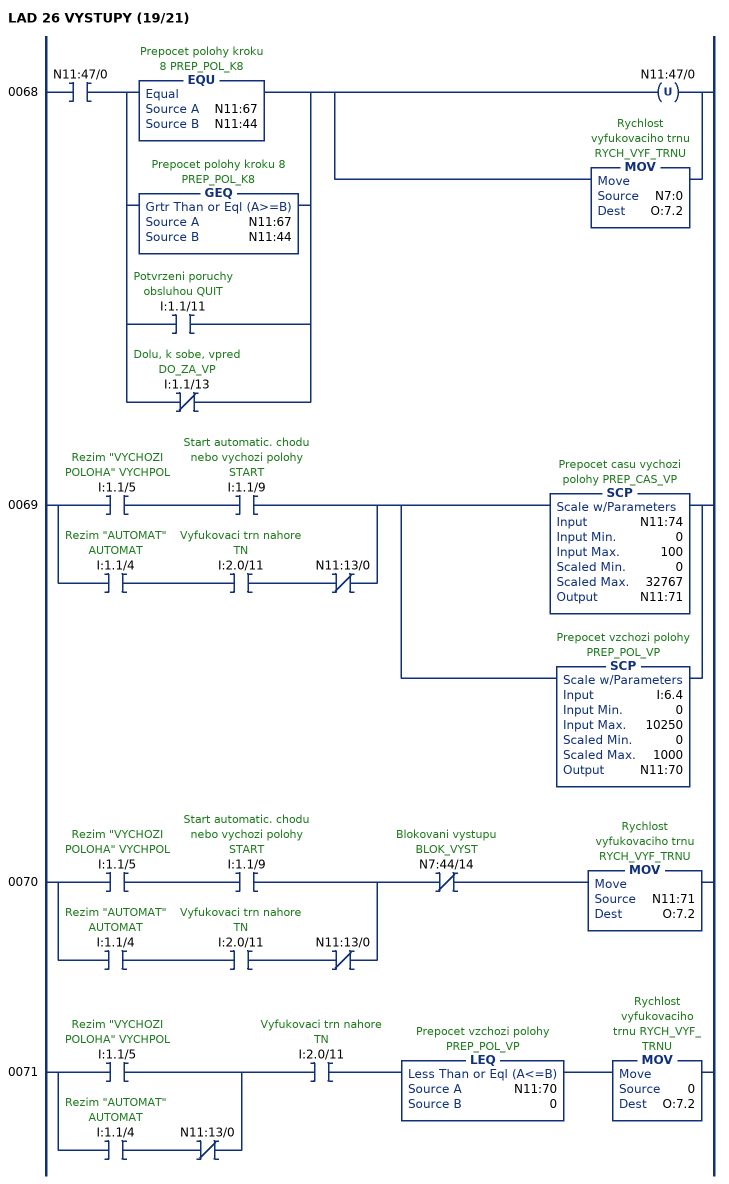
% Rung: 68 %
SOR XIC N11:47/0 BST EQU N11:67 N11:44 NXB GEQ N11:67 N11:44 NXB XIC I:1.1/11 NXB XIO I:1.1/13 BND BST OTU N11:47/0 NXB MOV N7:0 O:7.2 BND EOR
%   N11:67  PREP_POL_K8  "Prepocet polohy kroku 8" %
%   N11:44  DR_K8  "Draha kroku 8" %
%   I:1.1/11  QUIT  "Potvrzeni poruchy obsluhou" %
%   I:1.1/13  DO_ZA_VP  "Dolu, k sobe, vpred" %
%   O:7.2  RYCH_VYF_TRNU  "Rychlost vyfukovaciho trnu" %
% Rung: 69 %
SOR BST XIC I:1.1/5 XIC I:1.1/9 NXB XIC I:1.1/4 XIC I:2.0/11 XIO N11:13/0 BND BST SCP N11:74 0 100 0 32767 N11:71 NXB SCP I:6.4 0 10250 0 1000 N11:70 BND EOR
%   I:1.1/5  VYCHPOL  "Rezim "VYCHOZI POLOHA"" %
%   I:1.1/9  START  "Start automatic. chodu nebo vychozi polohy" %
%   I:1.1/4  AUTOMAT  "Rezim "AUTOMAT"" %
%   I:2.0/11  TN  "Vyfukovaci trn nahore" %
%   N11:74  CAS_VP %
%   N11:71  PREP_CAS_VP  "Prepocet casu vychozi polohy" %
%   I:6.4  POL_VYF_TRNU  "Poloha vyfukovaciho trnu" %
%   N11:70  PREP_POL_VP  "Prepocet vzchozi polohy" %
% Rung: 70 %
SOR BST XIC I:1.1/5 XIC I:1.1/9 NXB XIC I:1.1/4 XIC I:2.0/11 XIO N11:13/0 BND XIO N7:44/14 MOV N11:71 O:7.2 EOR
%   I:1.1/5  VYCHPOL  "Rezim "VYCHOZI POLOHA"" %
%   I:1.1/9  START  "Start automatic. chodu nebo vychozi polohy" %
%   I:1.1/4  AUTOMAT  "Rezim "AUTOMAT"" %
%   I:2.0/11  TN  "Vyfukovaci trn nahore" %
%   N7:44/14  BLOK_VYST  "Blokovani vystupu" %
%   N11:71  PREP_CAS_VP  "Prepocet casu vychozi polohy" %
%   O:7.2  RYCH_VYF_TRNU  "Rychlost vyfukovaciho trnu" %
% Rung: 71 %
SOR BST XIC I:1.1/5 NXB XIC I:1.1/4 XIO N11:13/0 BND XIC I:2.0/11 LEQ N11:70 0 MOV 0 O:7.2 EOR
%   I:1.1/5  VYCHPOL  "Rezim "VYCHOZI POLOHA"" %
%   I:1.1/4  AUTOMAT  "Rezim "AUTOMAT"" %
%   I:2.0/11  TN  "Vyfukovaci trn nahore" %
%   N11:70  PREP_POL_VP  "Prepocet vzchozi polohy" %
%   O:7.2  RYCH_VYF_TRNU  "Rychlost vyfukovaciho trnu" %

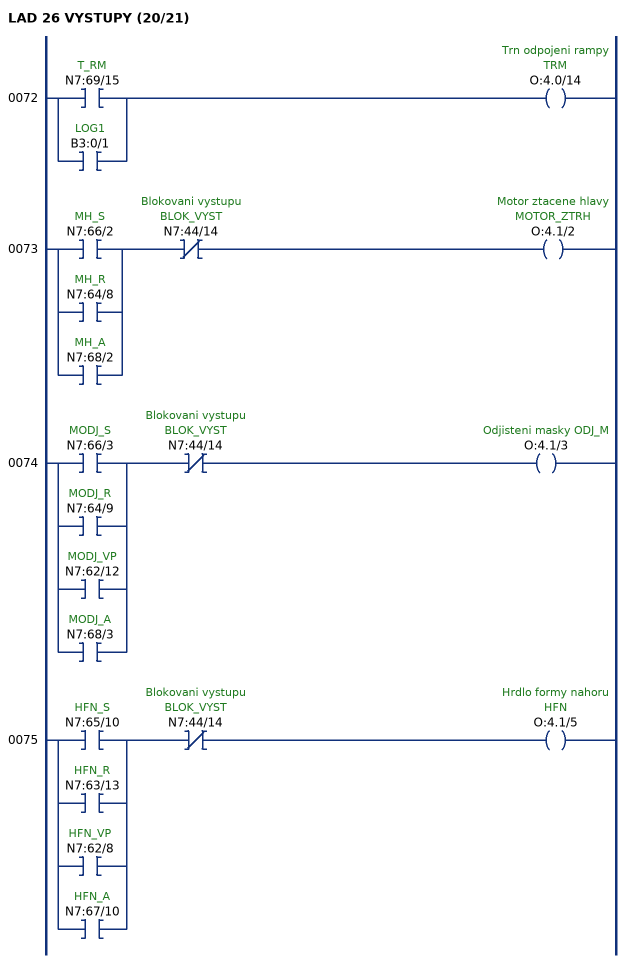
% Rung: 72 %
SOR BST XIC N7:69/15 NXB XIC B3:0/1 BND OTE O:4.0/14 EOR
%   N7:69/15  T_RM %
%   B3:0/1  LOG1 %
%   O:4.0/14  TRM  "Trn odpojeni rampy" %
% Rung: 73 %
SOR BST XIC N7:66/2 NXB XIC N7:64/8 NXB XIC N7:68/2 BND XIO N7:44/14 OTE O:4.1/2 EOR
%   N7:66/2  MH_S %
%   N7:64/8  MH_R %
%   N7:68/2  MH_A %
%   N7:44/14  BLOK_VYST  "Blokovani vystupu" %
%   O:4.1/2  MOTOR_ZTRH  "Motor ztacene hlavy" %
% Rung: 74 %
SOR BST XIC N7:66/3 NXB XIC N7:64/9 NXB XIC N7:62/12 NXB XIC N7:68/3 BND XIO N7:44/14 OTE O:4.1/3 EOR
%   N7:66/3  MODJ_S %
%   N7:64/9  MODJ_R %
%   N7:62/12  MODJ_VP %
%   N7:68/3  MODJ_A %
%   N7:44/14  BLOK_VYST  "Blokovani vystupu" %
%   O:4.1/3  ODJ_M  "Odjisteni masky" %
% Rung: 75 %
SOR BST XIC N7:65/10 NXB XIC N7:63/13 NXB XIC N7:62/8 NXB XIC N7:67/10 BND XIO N7:44/14 OTE O:4.1/5 EOR
%   N7:65/10  HFN_S %
%   N7:63/13  HFN_R %
%   N7:62/8  HFN_VP %
%   N7:67/10  HFN_A %
%   N7:44/14  BLOK_VYST  "Blokovani vystupu" %
%   O:4.1/5  HFN  "Hrdlo formy nahoru" %

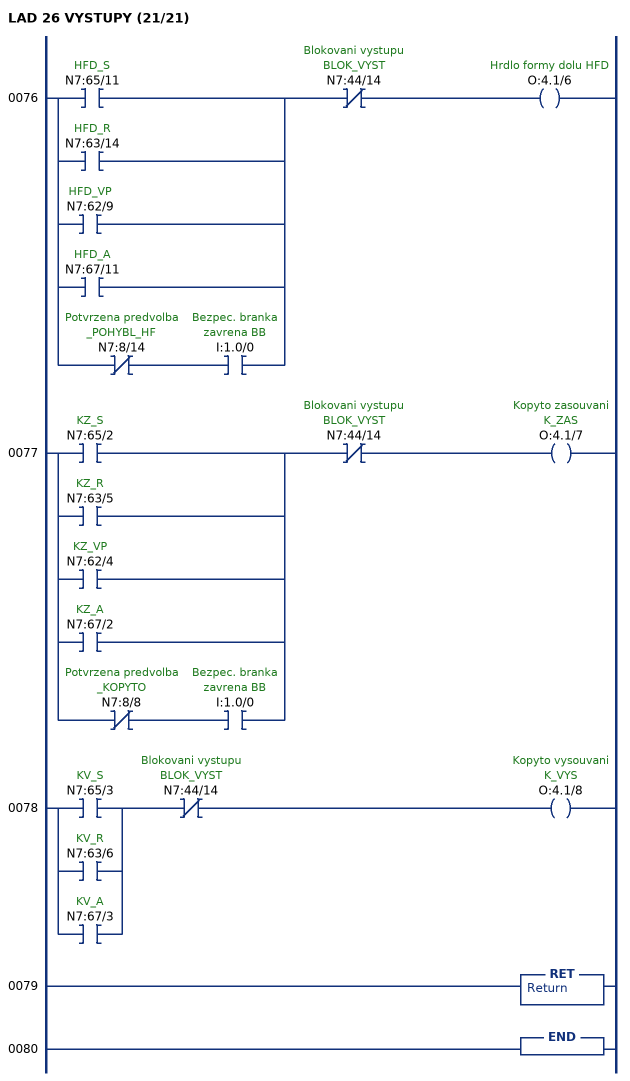
% Rung: 76 %
SOR BST XIC N7:65/11 NXB XIC N7:63/14 NXB XIC N7:62/9 NXB XIC N7:67/11 NXB XIO N7:8/14 XIC I:1.0/0 BND XIO N7:44/14 OTE O:4.1/6 EOR
%   N7:65/11  HFD_S %
%   N7:63/14  HFD_R %
%   N7:62/9  HFD_VP %
%   N7:67/11  HFD_A %
%   N7:8/14  _POHYBL_HF  "Potvrzena predvolba" %
%   I:1.0/0  BB  "Bezpec. branka zavrena" %
%   N7:44/14  BLOK_VYST  "Blokovani vystupu" %
%   O:4.1/6  HFD  "Hrdlo formy dolu" %
% Rung: 77 %
SOR BST XIC N7:65/2 NXB XIC N7:63/5 NXB XIC N7:62/4 NXB XIC N7:67/2 NXB XIO N7:8/8 XIC I:1.0/0 BND XIO N7:44/14 OTE O:4.1/7 EOR
%   N7:65/2  KZ_S %
%   N7:63/5  KZ_R %
%   N7:62/4  KZ_VP %
%   N7:67/2  KZ_A %
%   N7:8/8  _KOPYTO  "Potvrzena predvolba" %
%   I:1.0/0  BB  "Bezpec. branka zavrena" %
%   N7:44/14  BLOK_VYST  "Blokovani vystupu" %
%   O:4.1/7  K_ZAS  "Kopyto zasouvani" %
% Rung: 78 %
SOR BST XIC N7:65/3 NXB XIC N7:63/6 NXB XIC N7:67/3 BND XIO N7:44/14 OTE O:4.1/8 EOR
%   N7:65/3  KV_S %
%   N7:63/6  KV_R %
%   N7:67/3  KV_A %
%   N7:44/14  BLOK_VYST  "Blokovani vystupu" %
%   O:4.1/8  K_VYS  "Kopyto vysouvani" %
% Rung: 79 %
SOR RET EOR
% Rung: 80 %
SOR END EOR

LADDER 27 "REC_ARCHIV"
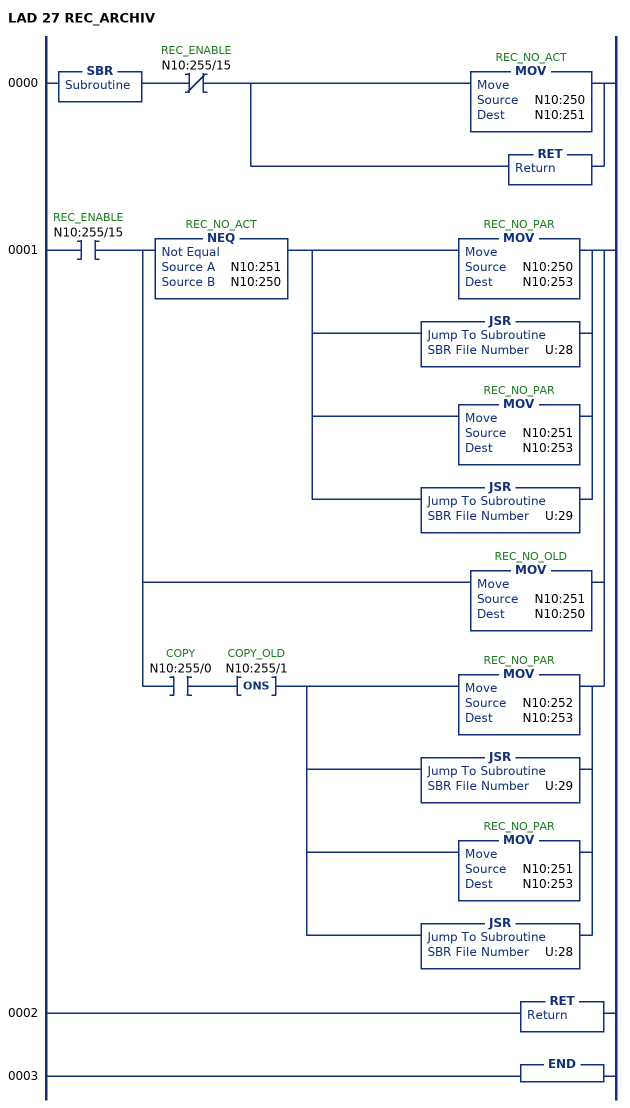
% Rung: 0 %
SOR SBR XIO N10:255/15 BST MOV N10:250 N10:251 NXB RET BND EOR
%   N10:255/15  REC_ENABLE %
%   N10:250  REC_NO_OLD %
%   N10:251  REC_NO_ACT %
% Rung: 1 %
SOR XIC N10:255/15 BST NEQ N10:251 N10:250 BST MOV N10:250 N10:253 NXB JSR U:28 NXB MOV N10:251 N10:253 NXB JSR U:29 BND NXB MOV N10:251 N10:250 NXB XIC N10:255/0 OSR N10:255/1 BST MOV N10:252 N10:253 NXB JSR U:29 NXB MOV N10:251 N10:253 NXB JSR U:28 BND BND EOR
%   N10:255/15  REC_ENABLE %
%   N10:251  REC_NO_ACT %
%   N10:250  REC_NO_OLD %
%   N10:253  REC_NO_PAR %
%   JSR U:28  "REC_SAVE" %
%   JSR U:29  "REC_LOAD" %
%   N10:255/0  COPY %
%   N10:255/1  COPY_OLD %
%   N10:252  REC_NO_SRC %
% Rung: 2 %
SOR RET EOR
% Rung: 3 %
SOR END EOR

LADDER 28 "REC_SAVE"
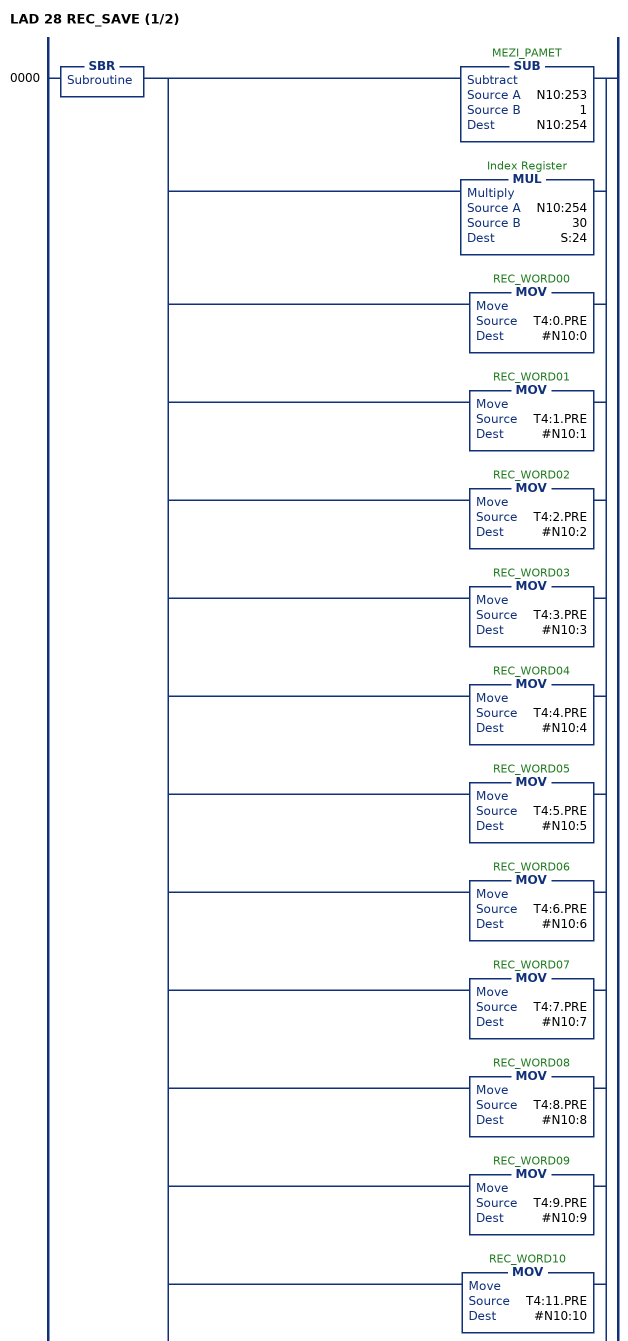
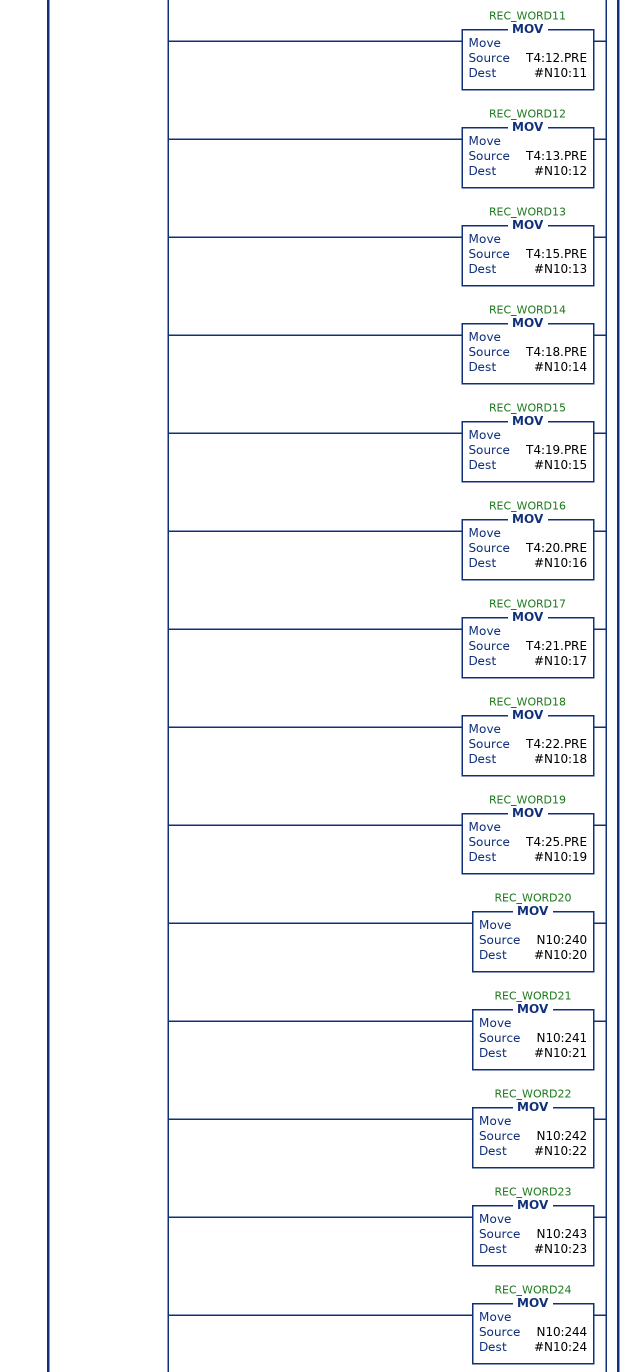
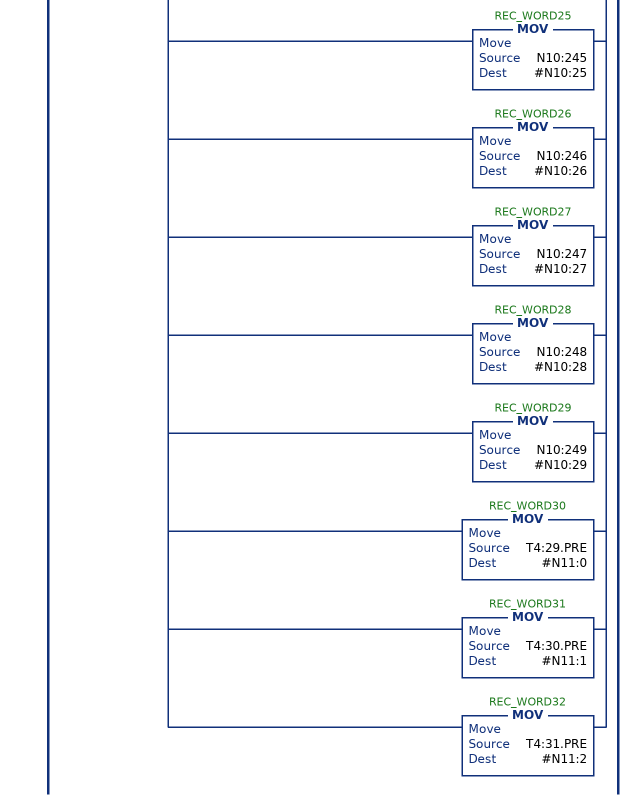
% Rung: 0 %
SOR SBR BST SUB N10:253 1 N10:254 NXB MUL N10:254 30 S:24 NXB MOV T4:0.PRE #N10:0 NXB MOV T4:1.PRE #N10:1 NXB MOV T4:2.PRE #N10:2 NXB MOV T4:3.PRE #N10:3 NXB MOV T4:4.PRE #N10:4 NXB MOV T4:5.PRE #N10:5 NXB MOV T4:6.PRE #N10:6 NXB MOV T4:7.PRE #N10:7 NXB MOV T4:8.PRE #N10:8 NXB MOV T4:9.PRE #N10:9 NXB MOV T4:11.PRE #N10:10 NXB MOV T4:12.PRE #N10:11 NXB MOV T4:13.PRE #N10:12 NXB MOV T4:15.PRE #N10:13 NXB MOV T4:18.PRE #N10:14 NXB MOV T4:19.PRE #N10:15 NXB MOV T4:20.PRE #N10:16 NXB MOV T4:21.PRE #N10:17 NXB MOV T4:22.PRE #N10:18 NXB MOV T4:25.PRE #N10:19 NXB MOV N10:240 #N10:20 NXB MOV N10:241 #N10:21 NXB MOV N10:242 #N10:22 NXB MOV N10:243 #N10:23 NXB MOV N10:244 #N10:24 NXB MOV N10:245 #N10:25 NXB MOV N10:246 #N10:26 NXB MOV N10:247 #N10:27 NXB MOV N10:248 #N10:28 NXB MOV N10:249 #N10:29 NXB MOV T4:29.PRE #N11:0 NXB MOV T4:30.PRE #N11:1 NXB MOV T4:31.PRE #N11:2 BND EOR
%   N10:253  REC_NO_PAR %
%   N10:254  MEZI_PAMET %
%   S:24  "Index Register" %
%   T4:0  PRODLEVA_1  "Prodleva po startu 1.cyklu" %
%   N10:0  REC_WORD00 %
%   T4:1  CAS_CYKLU  "Cas jednoho pracovniho cyklu stroje" %
%   N10:1  REC_WORD01 %
%   T4:2  ZAC_PVZ  "Zacatek podpurneho vzduchu" %
%   N10:2  REC_WORD02 %
%   T4:3  TRVANI_PVZ  "Trvani podpurneho vzduchu" %
%   N10:3  REC_WORD03 %
%   T4:4  KOPY_VPRED  "Kopyto nebo hlava vpred" %
%   N10:4  REC_WORD04 %
%   T4:5  KOPY_STOP  "Omezeni vysouvani kopyta" %
%   N10:5  REC_WORD05 %
%   T4:6  ZAC_VYFUK  "Zacatek vyfukovani" %
%   N10:6  REC_WORD06 %
%   T4:7  KONEC_VYF  "Konec vyfukovani" %
%   N10:7  REC_WORD07 %
%   T4:8  ODVETRANI  "Doba odvetrani nadoby" %
%   N10:8  REC_WORD08 %
%   T4:9  ZAC_ODDEL  "Zacatek oddelovani parizonu" %
%   N10:9  REC_WORD09 %
%   T4:11  SVAR_PARIZ  "Svarovani parizonu" %
%   N10:10  REC_WORD10 %
%   T4:12  VO_PO_DOLU  "Pomaly chod voziku shora" %
%   N10:11  REC_WORD11 %
%   T4:13  FORM_ZAVIR  "Zacatek zavirani formy pod vytl. hlavou" %
%   N10:12  REC_WORD12 %
%   T4:15  HF_NAHORU  "Hrdlo formy nahoru" %
%   N10:13  REC_WORD13 %
%   T4:18  ZAC_CO2 %
%   N10:14  REC_WORD14 %
%   T4:19  KON_CO2 %
%   N10:15  REC_WORD15 %
%   T4:20  PULZ_CO2 %
%   N10:16  REC_WORD16 %
%   T4:21  MEZ_CO2 %
%   N10:17  REC_WORD17 %
%   T4:22  KOP_VYSU  "Prodleva po vysunu- ti kopyta" %
%   N10:18  REC_WORD18 %
%   T4:25  FOR_OTVIRA  "Pomale otvirani formy" %
%   N10:19  REC_WORD19 %
%   N10:240  INF_TEMP01 %
%   N10:20  REC_WORD20 %
%   N10:241  INF_TEMP02 %
%   N10:21  REC_WORD21 %
%   N10:242  INF_TEMP03 %
%   N10:22  REC_WORD22 %
%   N10:243  INF_TEMP04 %
%   N10:23  REC_WORD23 %
%   N10:244  INF_TEMP05 %
%   N10:24  REC_WORD24 %
%   N10:245  INF_TEMP06 %
%   N10:25  REC_WORD25 %
%   N10:246  INF_TEMP07 %
%   N10:26  REC_WORD26 %
%   N10:247  INF_TEMP08 %
%   N10:27  REC_WORD27 %
%   N10:248  INF_BLOC64 %
%   N10:28  REC_WORD28 %
%   N10:249  INF_OT_VS %
%   N10:29  REC_WORD29 %
%   T4:29  PULZ_POT  "Doba oten potenciom. otek pohonu VS" %
%   N11:0  REC_WORD30 %
%   T4:30  PAR_NECLON  "Parizon nem zaclonit idlo" %
%   N11:1  REC_WORD31 %
%   T4:31  PAR_CLONIT  "Parizon m zaclonit idlo" %
%   N11:2  REC_WORD32 %

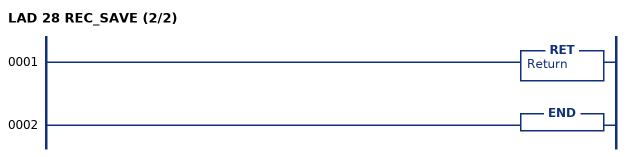
% Rung: 1 %
SOR RET EOR
% Rung: 2 %
SOR END EOR

LADDER 29 "REC_LOAD"
